{attribute 'linkalways'} 
{attribute 'no_explicit_call' := 'This FB is a CLASS and must be accessed using methods or properties'}
{attribute 'enable_dynamic_creation'}
FUNCTION_BLOCK Node_F_VN_SoftMax EXTENDS VisionNode
VAR
    ipSrcImage : _ITcVnImage;
    ipDestImage : _ITcVnImage;
    bFlatten : _BOOL(FALSE);
    hrPrev : _HRESULT(S_OK);
	hresult : _HRESULT(S_OK);
END_VAR

METHOD PUBLIC  Clone : I_Node
VAR
	pNode : POINTER TO Node_F_VN_SoftMax;
END_VAR
pNode := __NEW(Node_F_VN_SoftMax);
Clone := pNode^;
END_METHOD

METHOD FB_init : BOOL
VAR_INPUT
	bInitRetains : BOOL; // if TRUE, the retain variables are initialized (warm start / cold start)
	bInCopyCode : BOOL;  // if TRUE, the instance afterwards gets moved into the copy code (online change)
END_VAR
AddInput('ipSrcImage', ipSrcImage);
AddParameter('bFlatten', bFlatten);
AddInput('hrPrev', hrPrev);
AddOutput('ipDestImage', ipDestImage);
AddOutput('hresult',hresult);
END_METHOD

METHOD PROTECTED OnExecute
hresult.Value := F_VN_SoftMax(
    ipSrcImage := ipSrcImage.Value,
	ipDestImage := ipDestImage.Value,
    bFlatten := bFlatten.Value,
	hrPrev:= hrPrev.Value);
END_METHOD

METHOD PUBLIC PreExecutionCheck
VAR_INPUT
	Check : I_PreExecutionChecks;
END_VAR
Check.IsTrue(ipSrcImage.IsValid, 'ipSrcImage must contain an image');
Check.IsTrue(ipSrcImage.IsElementType(ETcVnElementType.TCVN_ET_REAL), 'ipSrcImage must be element type REAL');
Check.IsTrue(ipSrcImage.HasChannelCount(1), 'ipSrcImage must have 1 channel');
END_METHOD

END_FUNCTION_BLOCK

(* stored: Version 1.1.0.1, ProductVersion 3.1.4026.18
   POU Node_F_VN_SoftMax: Id {03f7d831-3fd7-0cf6-2f77-f02ea86089f4}, SpecialFunc None
   Folder Constructor: Id {d483c0ce-8d94-072f-0f37-7fbe1917ec8b}
   Method Clone: Id {016ee76e-a063-0399-33c2-5635ef8b25d0}
   Method FB_init: Id {b12a301d-b5cb-04f4-335e-ba26f0e72b89}
   Method OnExecute: Id {2faf220b-fc5f-0130-3ae4-149d705fa67c}
   Method PreExecutionCheck: Id {854ba822-6c86-0b59-258b-1c9fdf703fbe} *)
